TEXTLIST AxesMoveAlphaDeltaProcessUnitsTextList
  0 = 'd/m/s or h/m/s'
  1 = 'degrees'
  2 = 'arcmin'
  3 = 'arcsec'
  4 = 'rad'
   = ''
END_TEXTLIST

(* stored: Version 1.1.0.1, ProductVersion 3.1.4019.2
   TextList AxesMoveAlphaDeltaProcessUnitsTextList: Id {475472a6-25b3-4912-94ef-57dedd65349e} *)
